Fanuc KAREL source: kt00261.KL

-- PROVISIONAL review KL for V940-1; original PC SHA256 f04ed99626b6d787570fbdde24fe4b5095b11f5f5f8cedf9d4277ba9609ed1ea
-- Incomplete behavior may be omitted. Consult companion uncertainty JSON. Do not deploy.
PROGRAM KT00261
%NOLOCKGROUP
VAR
  R1 : REAL
  I2 : INTEGER
  OUT : BOOLEAN
BEGIN
  -- V9_ZERO_TABLE_METADATA_HINT layout=0001; no indexed target words; source/name/runtime held
  -- UNRESOLVED_PC offsets 5-16; opcodes 2E,23
  -- UNRESOLVED_PC offsets 21-32; opcodes 2E,23
  -- UNRESOLVED_PC offsets 37-57; opcodes 21,21,64,6D,23
  -- UNRESOLVED_PC offsets 62-66; opcodes 7F
END KT00261
